Universal Robots PolyScope program: husarion_ext_control.urp

Program husarion_ext_control (installation=default directory=/programs createdIn=5.13.1 lastSavedIn=5.13.1 robotSerialNumber=20235590039)
Calibrated DH parameters: a=[0.000132, -0.010838, -0.368353, 0.000022, 0.00001, 0]; d=[0.162671, 381.291062, -342.694886, -38.46257, 0.099751, 0.099545]; alpha=[1.569968, 0.001116, 0.00352, 1.570643, -1.571578, 0]; deltaTheta=[0, 1.545329, -1.191943, -0.353391, 0, 0]
InitVariablesNode
Robot Program (runOnlyOnce=false)
  URCap External Control (External Control, FZI Research Center for Information Technology)
